// TIA Portal V20 export
// export: Created 2025-12-01T14:57:26.4194698Z, ExportSetting None, DisplayName Totally Integrated Automation Portal, DisplayVersion V20 Update 3, DisplayName TIA Portal Openness, DisplayVersion V20 Update 3, DisplayName TIA Portal Version Control Interface, DisplayVersion V20 Update 3, DisplayName STEP 7 Professional, DisplayVersion V20 Update 3, DisplayName STEP 7 Safety, DisplayVersion V20 Update 2, DisplayName WinCC Basic/Comfort/Advanced, DisplayVersion V20 Update 3, DisplayName WinCC Professional, DisplayVersion V20 Update 3, DisplayName WinCC Unified, DisplayVersion V20 Update 3
DATA_BLOCK "DB600_ConfigQuimarox"   // DB600
{ S7_Optimized_Access := 'FALSE' }
// stored: AutoNumber false
   VAR RETAIN
      Quimarox : Array[1.."CTE_MaxNumQuimarox"] of Struct
         datos_config { S7_SetPoint := 'True'} : "CBS_Datos_config";
      END_STRUCT;
   END_VAR
BEGIN
   Quimarox[1].datos_config.Numero_MesaAsociada := 111;
   Quimarox[1].datos_config.Numero_vagones := 15;
   Quimarox[1].datos_config.Long_Vagon_mm := 1550;
   Quimarox[1].datos_config.Long_Util_vagon_mm := 1550;
   Quimarox[1].datos_config.dist_ini_vag_a_phs_mm := 1550;
   Quimarox[1].datos_config.maximo_encoder := DINT#2147483647;
   Quimarox[1].datos_config.relacion_mm_pulso := 2.187411;
END_DATA_BLOCK
